KUKA KRL program: InterconexEs.src

&ACCESS RV
&REL 3
&COMMENT INTERCONEXION ES
&USER
&PARAM EDITMASK = *
&PARAM TEMPLATE = C:\KRC\Roboter\Template\vorgabe
DEF InterconexEs( )
;################################################
; PROYECTO: MAFELEC PLANTA DE BATERIAS
; ROBOT: 121_R1
; PROGRAMA: INTERCONEXION SENALES A PLC EN SUBMIT
; CREADO POR: Alejandro Company(zaisor robotics)
; FECHA: 23-NOVIEMBRE-2022
; MODIFICADO POR:
; FECHA MODIFICACION: 17-DICIEMBRE-2022
;################################################


O_121R1S111B=I_121R1S111B
O_121R1S111A=I_121R1S111A
O_121R1S121B=I_121R1S121B
O_121R1S121A=I_121R1S121A
O_121R1S131B=I_121R1S131B
O_121R1S131A=I_121R1S131A
O_121R1S132B=I_121R1S132B
O_121R1S132A=I_121R1S132A
O_121R1S133B=I_121R1S133B
O_121R1S133A=I_121R1S133A
O_121R1S134B=I_121R1S134B
O_121R1S134A=I_121R1S134A
O_121R1S101=I_121R1S101
O_121R1S102=I_121R1S102
O_121R1S201=I_121R1S201
O_121R1S202=I_121R1S202
O_121R1S301=I_121R1S301
O_121R1S302=I_121R1S302
O_121R1S401=I_121R1S401
O_121R1S402=I_121R1S402
O_121R1S501=I_121R1S501
O_121R1S502=I_121R1S502
O_121R1S1000=I_121R1S1000

O_TYPE_INFO=I_TYPE_INFO

END
